ABB RobotStudio station: EGM_RWS_YuMi.rspag

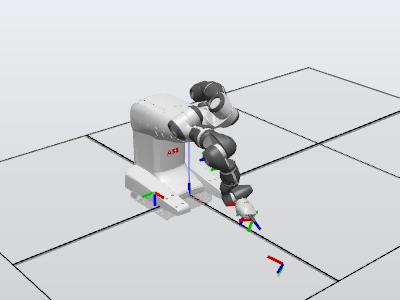
--- station ---
Station EGM_! (saved by RobotStudio 23.4.10609.1)
Controller EGM_1
  mechanical unit ROB_R: IRB14000_0.5_0.5_R, 6 joints, base frame (0, 0, 0) mm
  mechanical unit ROB_R_7: IRB14000_0.5_0.5_R, 1 joints, base frame (0, 0, 0) mm
  mechanical unit ROB_L: IRB14000_0.5_0.5_L, 6 joints, base frame (0, 0, 0) mm
  mechanical unit ROB_L_7: IRB14000_0.5_0.5_L, 1 joints, base frame (0, 0, 0) mm
Layout (positions relative to the parent item):
  - IRB14000_0.5_0.5 [mechanism, from %ABB.RobotStudio.Models.IRB14000%\IRB14000_0.5_0.5__02.rslib] at (0, 0, 0) mm
  - IRB14000_0.5_0.5_R [mechanism, from %ABB.RobotStudio.Models.IRB14000%\IRB14000_0.5_0.5__02.rslib] at (0, 0, 0) mm; joint values [-0.4135, 0.544, -0.0359, 0.2547, -2.9539, 1.6657, 1.0377] (rad or m)
  - IRB14000_0.5_0.5_L [mechanism, from %ABB.RobotStudio.Models.IRB14000%\IRB14000_0.5_0.5__02.rslib] at (0, 0, 0) mm; joint values [0, -2.2689, 2.3562, 0.5236, 0, 0.6981, 0] (rad or m)
  - Smart_Gripper_Servo_Camera_Fingers [mechanism, from %ABB.RobotStudio.Models.SmartGripper%\ABB_Smart_Gripper_Servo_Camera_Fingers.rslib] at (415.69, -21.05, 135.09) mm, rotated rx -102.54 ry -9.88 rz -102.72 deg; joint values [0] (rad or m)
  - Smart_Gripper_Servo_Camera_Fingers_2 [mechanism, from %ABB.RobotStudio.Models.SmartGripper%\ABB_Smart_Gripper_Servo_Camera_Fingers.rslib] at (-9.58, 182.61, 198.63) mm, rotated rx -179.34 ry -63.63 rz -15.45 deg; joint values [0] (rad or m)
Attachment: Smart_Gripper_Servo_Camera_Fingers is attached to IRB14000_0.5_0.5_R / Link7
Attachment: Smart_Gripper_Servo_Camera_Fingers_2 is attached to IRB14000_0.5_0.5_L / Link7
Targets, tools, work objects and paths stored in the station and not in the controller backup, written as RAPID:
! task T_ROB_R
MODULE EGM_IRB14000_test
  CONST robtarget move_r:=[[48.592406304,-256.414132391,126.402079594],[0,1,0,0],[0,2,-1,4],[-135,9E+09,9E+09,9E+09,9E+09,9E+09]];
  PROC Path_10()
    MoveJ Target_10,v1000,z100,tool0\WObj:=wobj0;
  ENDPROC
ENDMODULE

! task T_ROB_R
MODULE Module1
  CONST robtarget Target_20:=[[48.592667625,-256.414529528,126.402136711],[-0.000000037,1,0.000000057,-0.000000214],[0,2,-1,4],[-134.999970331,9E+09,9E+09,9E+09,9E+09,9E+09]];
ENDMODULE

! task T_ROB_R
MODULE CalibData
  PERS tooldata Servo:=[TRUE,[[0,0,114.2],[1,0,0,0]],[0.229,[7.9,12.4,48.7],[1,0,0,0],0.00021,0.00023,0.00008]];
  PERS tooldata Camera:=[TRUE,[[-7.3,28.3,35.1],[0.5,-0.5,0.5,0.5]],[0.229,[7.9,12.4,48.7],[1,0,0,0],0.00021,0.00023,0.00008]];
ENDMODULE

! task T_ROB_L
MODULE CalibData
  PERS tooldata Servo:=[TRUE,[[0,0,114.2],[1,0,0,0]],[0.229,[7.9,12.4,48.7],[1,0,0,0],0.00021,0.00023,0.00008]];
  PERS tooldata Camera:=[TRUE,[[-7.3,28.3,35.1],[0.5,-0.5,0.5,0.5]],[0.229,[7.9,12.4,48.7],[1,0,0,0],0.00021,0.00023,0.00008]];
ENDMODULE


--- Backups/EGM_1/HOME/EDS/EGM_Test_R/EGM_IRB14000_test.mod ---
MODULE EGM_IRB14000_test
    VAR egmident egmID;
    VAR egmstate egmSt1;
    CONST egm_minmax egm_minmax_joint1:=[-0.1,0.1];
    CONST egm_minmax egm_minmax_lin1:=[-1,1]; !in mm
    CONST egm_minmax egm_minmax_rot1:=[-2,2];! in degees
    ! For handling if the test is used with left or right arm.
    VAR jointtarget jpos10;
    VAR jointtarget joints;
    CONST jointtarget jpos10_L:=[[0,-130,30,0,40,0],[135,9E+09,9E+09,9E+09,9E+09,9E+09]];
    CONST jointtarget jpos10_R:=[[0,-130,30,0,40,0],[-135,9E+09,9E+09,9E+09,9E+09,9E+09]];
    CONST jointtarget JointTarget_1:=[[40,-120,3,-110,60,140],[-60,9E+09,9E+09,9E+09,9E+09,9E+09]]; !Created by Marie
    CONST jointtarget joints0 := [[0,0,0,0,0,0],[9E+09,9E+09,9E+09,9E+09,9E+09,9E+09]]; !Created by Marie

    PERS wobjdata Workobject_1:=[FALSE,TRUE,"",[[48.592406304,-256.414132391,126.402079594],[0,1,0,0]],[[0,0,0],[1,0,0,0]]];
    CONST robtarget Target_10:=[[48.592537483,-256.414332834,126.402138941],[0.000000131,1,0.000000039,-0.000000086],[0,2,-1,4],[-134.999969108,9E+09,9E+09,9E+09,9E+09,9E+09]];

    !PERS tooldata UISpenholder:=[TRUE,[[0,0,114.25],[1,0,0,0]],[1,[-0.095984607,0.082520613,38.69176324],[1,0,0,0],0,0,0]];
    VAR pose posecorTable:=[[150,-500,8],[1,0,0,0]];
    VAR pose posesenTable:=[[150,-500,8],[1,0,0,0]];

    ! Used tool
    TASK PERS tooldata
    tFroniusCMT:=[TRUE,[[12.3313,-0.108707,416.142],[0.903899,-0.00320735,0.427666,0.00765917]],[2.6,[-111.1,24.6,386.6],[1,0,0,0],0,0,0.072]];
    ! corr-frame: wobj, sens-frame: wobj
    TASK PERS wobjdata wobj_EGM1:=[FALSE,TRUE,"",[[150,1320,1140],[1,0,0,0]], [[0,0,0],[1,0,0,0]]];
    ! Correction frame offset: none
    VAR pose corr_frame_offs:=[[0,0,0],[1,0,0,0]];

    PROC main()
        ! Move to start position. Fine point is demanded.
        !MoveJ Target_10,v500,fine,tool0\WObj:=wobj0;
        !MoveAbsJ JointTarget_1,v1000,z100,tool0\WObj:=wobj0;  !Created by Marie
        StartMove;
        IF GetMecUnitName(ROB_ID) = "ROB_L" THEN
            !jpos10 := jpos10_L;
            !testAO;
            !stream;
            !testuc_UDP;
        ELSEIF GetMecUnitName(ROB_ID) = "ROB_R" THEN
            !jpos10 := jpos10_R;
            !testAO;
            !stream;
            testuc_UDP;
        ENDIF
    ENDPROC

    PROC StartMove()
        joints:=[[0,0,0,0,0,0],[9E+09,9E+09,9E+09,9E+09,9E+09,9E+09]];
        joints:=CjointT();
        IF joints=joints0 THEN
            TPErase;
            TPWrite "No Joints saved";
            Stop;
            ELSE
        MoveAbsJ joints, v500, fine, tool0;
        ENDIF
    ENDPROC

    PROC stream()
        EGMGetId egmID;
        EGMSetupAI ROB_ID, egmID, "default" \Pose \aiR1x:=ai_01
        \aiR2y:=ai_02 \aiR3z:=ai_04 \aiR4rx:=ai_05 \aiR5ry:=ai_06
        \aiR6rz:=ai_07 \aiE1:=ai_03;
        EGMActJoint egmID, \J1:=egm_minmax_joint1 \J3:=egm_minmax_joint1
        \J4:=egm_minmax_joint1;
        EGMRunJoint egmID, EGM_STOP_HOLD \J1 \J3 \RampInTime:=0.05;
    ENDPROC

    PROC testuc_UDP()
        EGMReset egmID;
        EGMGetId egmID;
        egmSt1 := EGMGetState(egmID);
        TPWrite "EGM state: "\Num := egmSt1;
        IF egmSt1 <= EGM_STATE_CONNECTED THEN
            ! Set up the EGM data source: UdpUc server using device "EGMsensor:"and configuration "default"
            !EGMSetupUC ROB_ID, egmID, "default", "EGMSensor" \Pose;
            EGMSetupUC ROB_ID, egmID, "default", "EGMSensor" \Joint; !Setup the UdpUc protocol for EGM joint control
        ENDIF
        runEGM;
        IF egmSt1 = EGM_STATE_CONNECTED THEN
            TPWrite "Reset EGM instance egmID";
            EGMReset egmID;
        ENDIF
    ENDPROC

    PROC runEGM()
        !EGMActPose egmID\Tool:=tool0, corr_frame_offs,EGM_FRAME_WORLD, tool0.tframe, EGM_FRAME_TOOL
        !\x:=egm_minmax_lin1 \y:=egm_minmax_lin1 \z:=egm_minmax_lin1
        !\rx:=egm_minmax_rot1 \ry:=egm_minmax_rot1 \rz:=egm_minmax_rot1 \LpFilter:=20;

        !EGMRunPose egmID, EGM_STOP_HOLD \x \y \z \CondTime:=20 \RampInTime:=0.05;

        EGMActJoint egmID, \J1:=egm_minmax_joint1 \J2:=egm_minmax_joint1 \J3:=egm_minmax_joint1
        \J4:=egm_minmax_joint1 \J5:=egm_minmax_joint1 \J6:=egm_minmax_joint1 \J7:=egm_minmax_joint1 ;

        EGMRunJoint egmID, EGM_STOP_HOLD \J1 \J2 \J3 \J4 \J5 \J6 \J7 \CondTime:=20 \RampInTime:=0.05;

        egmSt1:=EGMGetState(egmID);
    ENDPROC


    PROC testAO()
        ! Get an EGM idenity.
        EGMGetId egmID;
        ! Set up the EGM data source:
        ! Analog output signals and configuration "default".
        ! Only the EGM Joint mode support IRB14000.
        ! Notice the joint mapping of the analog output signals.
        EGMSetupAO ROB_ID, egmID, "default" \Pose \aoR1x:=ao_J1
        \aoR2y:=ao_J2 \aoR3z:=ao_J4 \aoR4rx:=ao_J5 \aoR5ry:=ao_J6
        \aoR6rz:=ao_J7 \AoE1:=ao_J3;
        ! Move to the starting point - fine point is needed.
        MoveAbsJ jpos10\NoEOffs, v50, fine, tool0;
        ! Set the signals (using an incrementing offset from the initial position).
        ! Another set of analog signals should be created, if running this code for both arms at the same time.
        ! Notice the joint mapping from a jointtarget to the analog output signals.
        SetAO ao_J1, jpos10.robax.rax_1 + 1;
        SetAO ao_J2, jpos10.robax.rax_2 + 2;
        SetAO ao_J3, jpos10.extax.eax_a + 3;
        SetAO ao_J4, jpos10.robax.rax_3 + 4;
        SetAO ao_J5, jpos10.robax.rax_4 + 5;
        SetAO ao_J6, jpos10.robax.rax_5 + 6;
        SetAO ao_J7, jpos10.robax.rax_6 + 7;
        ! Joint guidance for joints 1-7.
        EGMActJoint egmID \J1:=egm_minmax_joint1 \J2:=egm_minmax_joint1
        \J3:=egm_minmax_joint1 \J4:=egm_minmax_joint1
        \J5:=egm_minmax_joint1 \J6:=egm_minmax_joint1
        \J7:=egm_minmax_joint1 \LpFilter:=20;
        ! Run: keep the end position without returning to the start position.
        EGMRunJoint egmID, EGM_STOP_HOLD \J1 \J2 \J3 \J4 \J5 \J6 \J7
        \CondTime:=1 \RampInTime:=0.05 \PosCorrGain:=1;
        EGMReset egmID;

    ENDPROC
ENDMODULE

--- Backups/EGM_1/HOME/EDS/EGM_Test_R/Module1.mod ---
MODULE Module1
ENDMODULE

--- Backups/EGM_1/SYSPAR/EIO.cfg ---
EIO:CFG_1.0:6:1::
#
SYSSIG_OUT:

      -Status "MechUnitNotMoving" -Signal "OUTPUT_STATIONARY_ROB_L"\
      -Arg1 "ROB_L"

      -Status "MechUnitNotMoving" -Signal "OUTPUT_STATIONARY_ROB_R"\
      -Arg1 "ROB_R"
#
SYSSIG_IN:

      -Signal "Collision_Avoidance" -Action "CollAvoidance"
#
INDUSTRIAL_NETWORK:

      -Name "EtherNetIP" -Connection "Private Network" -Label "EtherNet/IP"

      -Name "DeviceNet" -Label "DeviceNet Master/Slave Network" -Address "2"
#
EIO_CROSS:

      -Name "Cross_Signal_Lamp" -Res "Signal_Lamp" -Act1 "DRV1BRAKE"
#
EIO_SIGNAL_SAFELEVEL:

      -Name "FlangePowerSafeLevel" -ActionWhenStartup "Last"

      -Name "SGcmdSafeLevel" -ActionWhenAccessible "Default"
#
ETHERNETIP_DEVICE:

      -Name "Hand_R" -VendorName "ABB" -ProductName "EtherNet/IP EIP" -Label "2"\
      -Address "192.168.125.30" -VendorId 75 -ProductCode 1 -OutputAssembly 100\
      -InputAssembly 101 -InputConnectionType "POINT2POINT" -OutputSize 10\
      -InputSize 10 -O2T_RPI 10000 -T2O_RPI 10000

      -Name "Hand_L" -VendorName "ABB" -ProductName "EtherNet/IP EIP" -Label "1"\
      -Address "192.168.125.40" -VendorId 75 -ProductCode 1 -OutputAssembly 100\
      -InputAssembly 101 -InputConnectionType "POINT2POINT" -OutputSize 10\
      -InputSize 10 -O2T_RPI 10000 -T2O_RPI 10000
#
DEVICENET_DEVICE:

      -Name "D652_10" -VendorName "ABB Robotics" -ProductName "24 VDC Unit"\
      -Address 10 -ProductCode 26 -DeviceType 7 -ConnectionType "COS"\
      -OutputSize 2 -InputSize 2
#
DEVICENET_INTERNAL_DEVICE:

      -Name "DN_Internal_Device" -VendorName "ABB Robotics"\
      -ProductName "DeviceNet Internal Slave Device"
#
ETHERNETIP_INTERNAL_DEVICE:

      -Name "EN_Internal_Device" -VendorName "ABB Robotics"\
      -ProductName "EtherNet/IP Internal Adapter Device"
#
EIO_SIGNAL:

      -Name "custom_DI_0" -SignalType "DI" -Device "D652_10" -DeviceMap "0"

      -Name "custom_DI_1" -SignalType "DI" -Device "D652_10" -DeviceMap "1"

      -Name "custom_DI_2" -SignalType "DI" -Device "D652_10" -DeviceMap "2"

      -Name "custom_DI_3" -SignalType "DI" -Device "D652_10" -DeviceMap "3"

      -Name "custom_DI_4" -SignalType "DI" -Device "D652_10" -DeviceMap "4"

      -Name "custom_DI_5" -SignalType "DI" -Device "D652_10" -DeviceMap "5"

      -Name "custom_DI_6" -SignalType "DI" -Device "D652_10" -DeviceMap "6"

      -Name "custom_DI_7" -SignalType "DI" -Device "D652_10" -DeviceMap "7"

      -Name "custom_DO_0" -SignalType "DO" -Device "D652_10" -DeviceMap "0"

      -Name "custom_DO_1" -SignalType "DO" -Device "D652_10" -DeviceMap "1"

      -Name "custom_DO_2" -SignalType "DO" -Device "D652_10" -DeviceMap "2"

      -Name "custom_DO_3" -SignalType "DO" -Device "D652_10" -DeviceMap "3"

      -Name "custom_DO_4" -SignalType "DO" -Device "D652_10" -DeviceMap "4"

      -Name "custom_DO_5" -SignalType "DO" -Device "D652_10" -DeviceMap "5"

      -Name "custom_DO_6" -SignalType "DO" -Device "D652_10" -DeviceMap "6"

      -Name "custom_DO_7" -SignalType "DO" -Device "D652_10" -DeviceMap "7"

      -Name "hall_sensor_joint_1" -SignalType "DI" -Device "D652_10"\
      -DeviceMap "8"

      -Name "hall_sensor_joint_2" -SignalType "DI" -Device "D652_10"\
      -DeviceMap "9"

      -Name "hall_sensor_joint_3" -SignalType "DI" -Device "D652_10"\
      -DeviceMap "11"

      -Name "hall_sensor_joint_4" -SignalType "DI" -Device "D652_10"\
      -DeviceMap "12"

      -Name "hall_sensor_joint_5" -SignalType "DI" -Device "D652_10"\
      -DeviceMap "13"

      -Name "hall_sensor_joint_6" -SignalType "DI" -Device "D652_10"\
      -DeviceMap "14"

      -Name "hall_sensor_joint_7" -SignalType "DI" -Device "D652_10"\
      -DeviceMap "10"

      -Name "hall_sensor_24V_ROB_R" -SignalType "DO" -Device "D652_10"\
      -DeviceMap "8"

      -Name "hall_sensor_24V_ROB_L" -SignalType "DO" -Device "D652_10"\
      -DeviceMap "9"

      -Name "flange_24V_ROB_R" -SignalType "DO" -Device "D652_10"\
      -DeviceMap "10" -SafeLevel "FlangePowerSafeLevel"

      -Name "flange_24V_ROB_L" -SignalType "DO" -Device "D652_10"\
      -DeviceMap "11" -SafeLevel "FlangePowerSafeLevel"

      -Name "Signal_Lamp" -SignalType "DO" -Device "D652_10" -DeviceMap "12"

      -Name "Collision_Avoidance" -SignalType "DO" -Access "All" -Default 1

      -Name "hand_CmdGripper_R" -SignalType "GO" -Device "Hand_R"\
      -Label "Hand Command Right" -DeviceMap "0-4" -Category "HandRight"\
      -Access "All" -SafeLevel "SGcmdSafeLevel"

      -Name "hand_CmdClearErr_R" -SignalType "DO" -Device "Hand_R"\
      -Label "Clear Error Right" -DeviceMap "7" -Category "HandRight"\
      -Access "All"

      -Name "hand_MaxPosition_R" -SignalType "GO" -Device "Hand_R"\
      -Label "Max Position Right" -DeviceMap "8-15" -Category "HandRight"\
      -Access "All" -Default 100

      -Name "hand_MinPosition_R" -SignalType "GO" -Device "Hand_R"\
      -Label "Min Position Right" -DeviceMap "16-23" -Category "HandRight"\
      -Access "All" -Default 50

      -Name "hand_MaxSpeed_R" -SignalType "GO" -Device "Hand_R"\
      -Label "Max Speed Right" -DeviceMap "24-31" -Category "HandRight"\
      -Access "All" -Default 200

      -Name "hand_HoldForce_R" -SignalType "GO" -Device "Hand_R"\
      -Label "Hold Force Right" -DeviceMap "40-47" -Category "HandRight"\
      -Access "All" -Default 120

      -Name "hand_CmdVacuum1_R" -SignalType "DO" -Device "Hand_R"\
      -Label "Vacuum 1 Right" -DeviceMap "48" -Category "HandRight"\
      -Access "All"

      -Name "hand_CmdVacuum2_R" -SignalType "DO" -Device "Hand_R"\
      -Label "Vacuum 2 Right" -DeviceMap "49" -Category "HandRight"\
      -Access "All"

      -Name "hand_CmdBlowoff1_R" -SignalType "DO" -Device "Hand_R"\
      -Label "BlowOff 1 Right" -DeviceMap "50" -Category "HandRight"\
      -Access "All"

      -Name "hand_CmdBlowoff2_R" -SignalType "DO" -Device "Hand_R"\
      -Label "BlowOff 2 Right" -DeviceMap "51" -Category "HandRight"\
      -Access "All"

      -Name "hand_SysState_R" -SignalType "GI" -Device "Hand_R"\
      -Label "Finger State Right" -DeviceMap "0-4" -Category "HandRight"\
      -Access "All"

      -Name "hand_SysError_R" -SignalType "GI" -Device "Hand_R"\
      -Label "Finger Error Right" -DeviceMap "32-39" -Category "HandRight"\
      -Access "All"

      -Name "hand_StatusCalibrated_R" -SignalType "DI" -Device "Hand_R"\
      -Label "Calibrated Right" -DeviceMap "5" -Category "HandRight"\
      -Access "All"

      -Name "hand_ActualPosition_R" -SignalType "GI" -Device "Hand_R"\
      -Label "Actual Position Right" -DeviceMap "8-15" -Category "HandRight"\
      -Access "All"

      -Name "hand_ActualSpeed_R" -SignalType "GI" -Device "Hand_R"\
      -Label "Actual Speed Right" -DeviceMap "16-23" -Category "HandRight"\
      -Access "All"

      -Name "hand_StatusCamLinked_R" -SignalType "DI" -Device "Hand_R"\
      -Label "Camera Connection Right" -DeviceMap "40" -Category "HandRight"\
      -Access "All"

      -Name "hand_SoftwareVersion_R" -SignalType "GI" -Device "Hand_R"\
      -Label "Software Version Right" -DeviceMap "41-47" -Category "HandRight"\
      -Access "All"

      -Name "hand_StatusVacuum1_R" -SignalType "DI" -Device "Hand_R"\
      -Label "Vacuum 1 Right Status" -DeviceMap "48" -Category "HandRight"\
      -Access "All"

      -Name "hand_StatusVacuum2_R" -SignalType "DI" -Device "Hand_R"\
      -Label "Vacuum 1 Right Status" -DeviceMap "49" -Category "HandRight"\
      -Access "All"

      -Name "hand_StatusBlowoff1_R" -SignalType "DI" -Device "Hand_R"\
      -Label "SuncTool 1 Right Status" -DeviceMap "50" -Category "HandRight"\
      -Access "All"

      -Name "hand_StatusBlowoff2_R" -SignalType "DI" -Device "Hand_R"\
      -Label "SuncTool 1 Right Status" -DeviceMap "51" -Category "HandRight"\
      -Access "All"

      -Name "hand_ActualPressure1_R" -SignalType "GI" -Device "Hand_R"\
      -Label "Vacuum pressure1 Right" -DeviceMap "64-71" -Category "HandRight"\
      -Access "All"

      -Name "hand_ActualPressure2_R" -SignalType "GI" -Device "Hand_R"\
      -Label "Vacuum pressure2 Right" -DeviceMap "72-79" -Category "HandRight"\
      -Access "All"

      -Name "hand_SecurityKey_R" -SignalType "GO" -Device "Hand_R"\
      -Label "Security key right" -DeviceMap "64-71" -Category "HandRight"\
      -Access "All"

      -Name "hand_TftPFtpMode_R" -SignalType "DI" -Device "Hand_R"\
      -Label "Hand firmware update mode" -DeviceMap "7" -Category "HandRight"\
      -Access "All"

      -Name "hand_CmdGripper_L" -SignalType "GO" -Device "Hand_L"\
      -Label "Hand Command Left" -DeviceMap "0-4" -Category "HandLeft"\
      -Access "All" -SafeLevel "SGcmdSafeLevel"

      -Name "hand_CmdClearErr_L" -SignalType "DO" -Device "Hand_L"\
      -Label "Clear Error Left" -DeviceMap "7" -Category "HandLeft"\
      -Access "All"

      -Name "hand_MaxPosition_L" -SignalType "GO" -Device "Hand_L"\
      -Label "Max Position Left" -DeviceMap "8-15" -Category "HandLeft"\
      -Access "All" -Default 100

      -Name "hand_MinPosition_L" -SignalType "GO" -Device "Hand_L"\
      -Label "Min Position Left" -DeviceMap "16-23" -Category "HandLeft"\
      -Access "All" -Default 50

      -Name "hand_MaxSpeed_L" -SignalType "GO" -Device "Hand_L"\
      -Label "Max Speed Left" -DeviceMap "24-31" -Category "HandLeft"\
      -Access "All" -Default 200

      -Name "hand_HoldForce_L" -SignalType "GO" -Device "Hand_L"\
      -Label "Hold Force Left" -DeviceMap "40-47" -Category "HandLeft"\
      -Access "All" -Default 120

      -Name "hand_CmdVacuum1_L" -SignalType "DO" -Device "Hand_L"\
      -Label "Vacuum 1 Left" -DeviceMap "48" -Category "HandLeft" -Access "All"

      -Name "hand_CmdVacuum2_L" -SignalType "DO" -Device "Hand_L"\
      -Label "Vacuum 2 Left" -DeviceMap "49" -Category "HandLeft" -Access "All"

      -Name "hand_CmdBlowoff1_L" -SignalType "DO" -Device "Hand_L"\
      -Label "BlowOff 1 Left" -DeviceMap "50" -Category "HandLeft" -Access "All"

      -Name "hand_CmdBlowoff2_L" -SignalType "DO" -Device "Hand_L"\
      -Label "BlowOff 2 Left" -DeviceMap "51" -Category "HandLeft" -Access "All"

      -Name "hand_SysState_L" -SignalType "GI" -Device "Hand_L"\
      -Label "Finger State Left" -DeviceMap "0-4" -Category "HandLeft"\
      -Access "All"

      -Name "hand_SysError_L" -SignalType "GI" -Device "Hand_L"\
      -Label "Finger Error Left" -DeviceMap "32-39" -Category "HandLeft"\
      -Access "All"

      -Name "hand_StatusCalibrated_L" -SignalType "DI" -Device "Hand_L"\
      -Label "Calibrated Left" -DeviceMap "5" -Category "HandLeft" -Access "All"

      -Name "hand_ActualPosition_L" -SignalType "GI" -Device "Hand_L"\
      -Label "Actual Position Left" -DeviceMap "8-15" -Category "HandLeft"\
      -Access "All"

      -Name "hand_ActualSpeed_L" -SignalType "GI" -Device "Hand_L"\
      -Label "Actual Speed Left" -DeviceMap "16-23" -Category "HandLeft"\
      -Access "All"

      -Name "hand_StatusCamLinked_L" -SignalType "DI" -Device "Hand_L"\
      -Label "Camera Connection Left" -DeviceMap "40" -Category "HandLeft"\
      -Access "All"

      -Name "hand_SoftwareVersion_L" -SignalType "GI" -Device "Hand_L"\
      -Label "Software Version Left" -DeviceMap "41-47" -Category "HandLeft"\
      -Access "All"

      -Name "hand_StatusVacuum1_L" -SignalType "DI" -Device "Hand_L"\
      -Label "Vacuum 1 Left Status" -DeviceMap "48" -Category "HandLeft"\
      -Access "All"

      -Name "hand_StatusVacuum2_L" -SignalType "DI" -Device "Hand_L"\
      -Label "Vacuum 1 Left Status" -DeviceMap "49" -Category "HandLeft"\
      -Access "All"

      -Name "hand_StatusBlowoff1_L" -SignalType "DI" -Device "Hand_L"\
      -Label "SuncTool 1 Left Status" -DeviceMap "50" -Category "HandLeft"\
      -Access "All"

      -Name "hand_StatusBlowoff2_L" -SignalType "DI" -Device "Hand_L"\
      -Label "SuncTool 1 Left Status" -DeviceMap "51" -Category "HandLeft"\
      -Access "All"

      -Name "hand_ActualPressure1_L" -SignalType "GI" -Device "Hand_L"\
      -Label "Vacuum pressure1 Left" -DeviceMap "64-71" -Category "HandLeft"\
      -Access "All"

      -Name "hand_ActualPressure2_L" -SignalType "GI" -Device "Hand_L"\
      -Label "Vacuum pressure2 Left" -DeviceMap "72-79" -Category "HandLeft"\
      -Access "All"

      -Name "hand_SecurityKey_L" -SignalType "GO" -Device "Hand_L"\
      -Label "Security key Left" -DeviceMap "64-71" -Category "HandLeft"\
      -Access "All"

      -Name "hand_TftPFtpMode_L" -SignalType "DI" -Device "Hand_L"\
      -Label "Hand firmware update mode" -DeviceMap "7" -Category "HandLeft"\
      -Access "All"

      -Name "RUN_RAPID_ROUTINE" -SignalType "DI" -Access "All"

      -Name "EGM_START_JOINT" -SignalType "DI" -Access "All"

      -Name "EGM_START_POSE" -SignalType "DI" -Access "All"

      -Name "EGM_STOP" -SignalType "DI" -Access "All"

      -Name "EGM_START_STREAM" -SignalType "DI" -Access "All"

      -Name "EGM_STOP_STREAM" -SignalType "DI" -Access "All"

      -Name "RUN_SG_ROUTINE" -SignalType "DI" -Access "All"

      -Name "OUTPUT_STATIONARY_ROB_L" -SignalType "DO" -Access "ReadOnly"

      -Name "OUTPUT_STATIONARY_ROB_R" -SignalType "DO" -Access "ReadOnly"
